TYPE E_MoveCmd :
(
	eCmd_Idle,
	eCmd_MoveAbsolute,
	eCmd_MoveModulo,
	eCmd_MoveRelative,
	eCmd_MoveVelocity
);
END_TYPE

(* stored: Version 1.1.0.1, ProductVersion 3.1.4024.11
   DUT E_MoveCmd: Id {b9de3213-fce6-4229-ac80-f4d5fa24c44b} *)
